(*
SPDX-FileCopyrightText: © 2026 Oleksandr Tiutyk <trofimich@gmail.com>
SPDX-License-Identifier: MIT
License: https://opensource.org/license/mit
*)

{attribute 'no_explicit_call' := 'do not call this function block directly'}
FUNCTION_BLOCK HmiTrafficLight EXTENDS TOF_Automation.HmiAutomationComponentElement
VAR_OUTPUT
	Statuses : HMI_TRAFFIC_LIGHT_STATUSES;
END_VAR
VAR_STAT
	//! <summary>Class name shared by all instances of this function block.</summary>
	{attribute 'hide'} 
	_ClassName : STRING := __POUNAME();
END_VAR

{attribute 'monitoring' := 'call'}
PROPERTY ClassName : REFERENCE TO STRING
GET
ClassName REF= _ClassName;
END_GET
END_PROPERTY

{attribute 'monitoring' := 'call'}
PROPERTY NamespaceName : REFERENCE TO STRING
GET
NamespaceName REF= CurrentNamespace.Name;
END_GET
END_PROPERTY

METHOD INTERNAL ProcessCommands
VAR_INPUT
	trafficLight : IReadOnlyTrafficLight;
END_VAR
ProcessAutomationComponentCommands(automationComponent := trafficLight);
END_METHOD

METHOD INTERNAL UpdateStatuses
VAR_INPUT
	trafficLight : IReadOnlyTrafficLight;
END_VAR
UpdateAutomationComponentStatuses(automationComponent := trafficLight);

Statuses.RedLightIsActive := trafficLight.RedLight.Value;
Statuses.YellowLightIsActive := trafficLight.YellowLight.Value;	
Statuses.GreenLightIsActive := trafficLight.GreenLight.Value;
END_METHOD

END_FUNCTION_BLOCK

(* stored: Version 1.1.0.1
   POU HmiTrafficLight: Id {441b1406-cc89-41ff-a025-db174ebf455b}, SpecialFunc None
   Property ClassName: Id {35032083-5d21-4bfc-a78d-caea3254f36f}
   Get Get: Id {07cbad6f-2f34-46d1-9f77-ae646fa2e39d}
   Property NamespaceName: Id {e0159771-ec48-495b-b532-34c13f690f68}
   Get Get: Id {28ae13a2-31bc-4689-b3b5-2be40a7b9975}
   Method ProcessCommands: Id {e63808dd-3cc3-43be-ac55-379611ff4ca2}
   Method UpdateStatuses: Id {6ea57841-67d8-4121-88dd-1fbb7ac6ce1e} *)
